VAR_GLOBAL

	iState : DINT; // My machine state.
	bStartButton : BOOL;
	
	arrPizzaHistory : ARRAY [0..100] OF ST_PIZZA;
	
	fbNT_GetTime : NT_GetTime;
	stCurrentTime : TIMESTRUCT;
	dtCurrentTime : DT;
END_VAR

(* stored: Version 1.1.0.1, ProductVersion 3.1.0.26
   GVL HMI_VARS: Id {15fd23c2-3235-4673-b77e-e3e929f0cb33} *)
